(* CoDeSys 2.3 export: STAPE.EXP *)

(* Data type in Other *)
TYPE StAPE:
(
    Wait:=0,
    WarmTank,
    WarmBath,
    FillFromTank,
    US,
    FiltrToTank,
    DrainToTank,
    FillFromNet,
    US2,
    FiltrToNet,
    DrainToNet,
    FillTank,
    ManToNet,
    ManToTank,
    Skip,
    Barb,
    Barb_and_Filtr,
    Dry,
    DeGas,
    Warning,
    Pump,
	Cooling,
	Heating
);
END_TYPE
